FUNCTION_BLOCK FB_CleaningProcessStateCleaning EXTENDS FB_CleaningProcessStateBase
VAR_INPUT
END_VAR

VAR_OUTPUT
END_VAR

VAR
END_VAR

METHOD mCleaningOp : BOOL
VAR_INPUT
	sI_Operation : EN_CLEANING_OP;
END_VAR
//Set mode and start process when successful
(*HOA TEST
IF NOT bL_DevOpActive THEN
  bL_DevOpActive := I_ParentCallback.mSetMode(sI_Operation);
  mCleaningOp    := TRUE; //report success
END_IF*) mCleaningOp    := TRUE;

//Switch to production mode if no operation active
IF I_MachineStatus.pSafetyOk AND I_MachineStatus.pMachineReady AND NOT bL_DevOpActive THEN
  IF sI_Operation = eOPCAPENTER THEN
    I_ParentCallback.mChangeState(EN_Cleaning_State.Capping);
  ELSIF sI_Operation = eOPCAPEXIT THEN
    I_ParentCallback.mChangeState(EN_Cleaning_State.CappingExit);
  ELSIF sI_Operation = eOPCLEAN THEN
    I_ParentCallback.mChangeState(EN_Cleaning_State.Cleaning);
  ELSIF sI_Operation = eOPPURGE THEN
    I_ParentCallback.mChangeState(EN_Cleaning_State.Capping);
  END_IF
END_IF
END_METHOD

METHOD mEntryAction
VAR_INPUT
END_VAR
iL_CurrentStep := 0;

// Launch initial command to bring system to service mode
bL_DevOpActive := I_ParentCallback.mSetMode(EN_CLEANING_OP.eOPCLEAN);
END_METHOD

METHOD mProduction : BOOL
VAR_INPUT
END_VAR
//Switch to production mode if no operation active
IF I_MachineStatus.pSafetyOk AND I_MachineStatus.pMachineReady AND NOT bL_DevOpActive THEN
	I_ParentCallback.mChangeState(EN_Cleaning_State.Production);
END_IF
END_METHOD

METHOD mService : BOOL
VAR_INPUT
END_VAR
//Switch to service mode
IF NOT bL_DevOpActive THEN
	I_ParentCallback.mChangeState(EN_Cleaning_State.Service);
END_IF
END_METHOD

METHOD mStateAction
VAR_INPUT
END_VAR
IF bL_DevOpActive THEN
	mDevOp();
END_IF

SUPER^.pInitDone := TRUE;
END_METHOD

END_FUNCTION_BLOCK

(* stored: Version 1.1.0.1, ProductVersion 3.1.4024.11
   POU FB_CleaningProcessStateCleaning: Id {e7c255d2-1d76-49d7-86a6-e8fb74668801}, SpecialFunc None
   Method mCleaningOp: Id {5668cd6a-884f-4852-8893-d6f52428e76e}
   Method mEntryAction: Id {2d6c324e-5819-43e8-89eb-c595bfd1967d}
   Method mProduction: Id {7d2da4d2-928d-464a-9983-9874a31b7aa0}
   Method mService: Id {4db18a26-0c97-4ca5-a0b7-58c6a18fb534}
   Method mStateAction: Id {c576a14c-236b-4577-9ab6-ebfcfd974a67} *)
